FUNCTION_BLOCK FB_SetRobotTM
VAR_INPUT
	cmdID : E_CommandEventTM;
	fX : REAL := 0; 
	fY : REAL := 0; 
	fZ : REAL := 0; 
	fRX : REAL := 0; 
	fRY : REAL := 0; 
	fRZ : REAL := 0; 
	
	fTheta1 : REAL := 0;
	fTheta2 : REAL := 0;
	fTheta3 : REAL := 0;
	fTheta4 : REAL := 0;
	fTheta5 : REAL := 0;
	fTheta6 : REAL := 0;
END_VAR
VAR_OUTPUT
END_VAR
VAR	
	arrTemp : ARRAY [0..1] OF WORD;
	eSetState : E_RobotStateTM := READY;
	
	//Modbus variables
    fbWrite16			: FB_MBWriteRegs;
	fbWrite6 			: FB_MBWriteSingleReg;
	bStart6 			: BOOL;
	bStart16 			: BOOL;
	arrWriteCommands 	: ARRAY [0..11] OF WORD;
	nQuantity			: WORD := INT_TO_WORD(SIZEOF(arrWriteCommands)/2);
	nMBAddr				: WORD; 
	bBusy6				: BOOL;
	bError6				: BOOL;
	nErrId6				: UDINT;
	bBusy16				: BOOL;
	bError16			: BOOL;
	nErrId16			: UDINT;
	sIPAddr				: STRING(15) := GCL_ModbusTcp.cIPAddr;
	nTCPPort			: UINT := GCL_ModbusTcp.cTCPPort;
	nUnitID				: BYTE := GCL_ModbusTcp.cUnitID;
	nValue				: WORD;
END_VAR


CASE eSetState OF
	READY:
		IF fbWrite6.bBusy THEN
			RETURN;
		END_IF
		eSetState := PREPARE;
		
	PREPARE:
		CASE cmdID OF 
			RobotHome: Home();
			MoveCartesianPTP: MoveRelPTP();
			SetJointPositions: SetJoints();
				
			SetJointSpeeds:
				nValue := 2#0000000000000011; // 3
				nMBAddr := 16#1B59;
			GripON:
				nValue := 2#0000000000000100; // 4
				nMBAddr := 16#1B59;
			GripOFF:
				nValue := 2#0000000000000101; // 5
				nMBAddr := 16#1B59;
				
		END_CASE
		eSetState := SEND;
		
	SEND:
		IF NOT bstart6 THEN	
			bStart6 := TRUE;
			fbWrite6.bExecute := TRUE;
		ELSE
			IF NOT fbWrite6.bBUSY THEN
				bStart6 := FALSE;
			END_IF
			fbWrite6.bExecute := FALSE;
		END_IF
		fbWrite6(sIPAddr:= sIPAddr, nTCPPort:= nTCPPort, nUnitID:= nUnitID, nMBAddr:= 16#23F0, nValue:=nValue,
				tTimeout:= T#1S, bBusy=>bBusy6, bError=> bError6, nErrId=> nErrId6 );
			
		IF NOT bStart16 THEN
			bStart16 := TRUE;
			fbWrite16.bExecute := TRUE;
		ELSE
			IF NOT fbWrite16.bBusy THEN
				bStart16 := FALSE;
			END_IF
			fbWrite16.bExecute := FALSE;
		END_IF
		
		fbWrite16(sIPAddr:= sIPAddr, nTCPPort:= nTCPPort, nUnitID:= nUnitID, nQuantity:= nQuantity, nMBAddr:= nMBAddr, cbLength:= SIZEOF(arrWriteCommands) , 
				pSrcAddr:= ADR(arrWriteCommands), bExecute:= bStart16 , tTimeout:= T#1S, bBusy=>bBusy16, bError=> bError16, nErrId=> nErrId16 );
		
		eSetState := READY;		
	
		
END_CASE

METHOD Home : BOOL
VAR_INPUT
END_VAR

//prepare the data to be sent 
nValue := 2#0000000000000000; // 0
nMBAddr := 16#23F1; //9201
END_METHOD

METHOD MoveRelPTP : BOOL
VAR_INPUT
END_VAR
// prepare

// e.g. next state := MoveRelPTP

//prepare the next state
eSetState := Send;

//prepare the data to be sent 
nValue := 2#0000000000000001; // 1
nMBAddr := 16#23F1; //9201

MEMCPY(ADR(arrTemp), ADR(fX), 4); //xPos
arrWriteCommands[0] := arrTemp[1];
arrWriteCommands[1] := arrTemp[0];

MEMCPY(ADR(arrTemp), ADR(fY), 4); //yPos
arrWriteCommands[2] := arrTemp[1];
arrWriteCommands[3] := arrTemp[0];

MEMCPY(ADR(arrTemp), ADR(fZ), 4); //zPos
arrWriteCommands[4] := arrTemp[1];
arrWriteCommands[5] := arrTemp[0];

MEMCPY(ADR(arrTemp), ADR(fRX), 4); //xRot
arrWriteCommands[6] := arrTemp[1];
arrWriteCommands[7] := arrTemp[0];

MEMCPY(ADR(arrTemp), ADR(fRY), 4); //yRot
arrWriteCommands[8] := arrTemp[1];
arrWriteCommands[9] := arrTemp[0];

MEMCPY(ADR(arrTemp), ADR(fRZ), 4); //zRot
arrWriteCommands[10] := arrTemp[1];
arrWriteCommands[11] := arrTemp[0];
END_METHOD

METHOD SetJoints : BOOL
VAR_INPUT
END_VAR
//prepare data to be sent 
nValue := 2#0000000000000010; // 2
nMBAddr := 16#23FC; //9212


MEMCPY(ADR(arrTemp), ADR(fTheta1), 4); // joint 1
arrWriteCommands[0] := arrTemp[1];
arrWriteCommands[1] := arrTemp[0];

MEMCPY(ADR(arrTemp), ADR(fTheta2), 4); // joint 2
arrWriteCommands[2] := arrTemp[1];
arrWriteCommands[3] := arrTemp[0];

MEMCPY(ADR(arrTemp), ADR(fTheta3), 4); // joint 3
arrWriteCommands[4] := arrTemp[1];
arrWriteCommands[5] := arrTemp[0];

MEMCPY(ADR(arrTemp), ADR(fTheta4), 4); // joint 4
arrWriteCommands[6] := arrTemp[1];
arrWriteCommands[7] := arrTemp[0];

MEMCPY(ADR(arrTemp), ADR(fTheta5), 4); // joint 5
arrWriteCommands[8] := arrTemp[1];
arrWriteCommands[9] := arrTemp[0];

MEMCPY(ADR(arrTemp), ADR(fTheta6), 4); // joint 6
arrWriteCommands[10] := arrTemp[1];
arrWriteCommands[11] := arrTemp[0];
END_METHOD

END_FUNCTION_BLOCK

(* stored: Version 1.1.0.1, ProductVersion 3.1.4024.11
   POU FB_SetRobotTM: Id {634abb87-82fc-4c2c-a846-4f9fa090629c}, SpecialFunc None
   Method Home: Id {845fdaf6-43f5-47d2-a9d1-62cdb2425f69}
   Method MoveRelPTP: Id {b2e16968-d0b3-4e43-a8fe-54226ace325e}
   Method SetJoints: Id {4d06ccc0-5e3f-4f8e-9775-089a6f900979} *)
